{attribute 'qualified_only'}
{attribute 'strict'}
TYPE E_LogFileSplitMode :
(
	eDontSplit := 0,
	eSplitByDay := 1,
	eSplitByHour := 2
);
END_TYPE

(* stored: Version 1.1.0.1, ProductVersion 3.1.4024.12
   DUT E_LogFileSplitMode: Id {69b546ef-1376-4ace-8c18-339749d44102} *)
